FUNCTION_BLOCK ResetTrigger
  (* Standard: 61499-2 *)
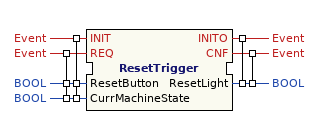
  EVENT_INPUT
    INIT WITH ResetButton, CurrMachineState;
    REQ WITH ResetButton, CurrMachineState;
  END_EVENT
  EVENT_OUTPUT
    INITO WITH ResetLight;
    CNF WITH ResetLight;
  END_EVENT
  VAR_INPUT
    ResetButton : BOOL;
    CurrMachineState : BOOL;
  END_VAR
  VAR_OUTPUT
    ResetLight : BOOL;
  END_VAR
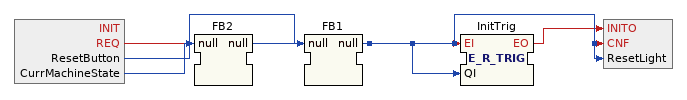
  FBS
    InitTrig : E_R_TRIG;
    FB1 : ;
    FB2 : ;
  END_FBS
  EVENT_CONNECTIONS
    FB1.null TO InitTrig.EI;
    FB2.null TO FB1.null;
    REQ TO FB2.null;
    InitTrig.EO TO INITO;
    FB1.null TO CNF;
  END_CONNECTIONS
  DATA_CONNECTIONS
    FB1.null TO InitTrig.QI;
    FB2.null TO FB1.null;
    FB1.null TO ResetLight;
    ResetButton TO FB1.null;
    CurrMachineState TO FB2.null;
  END_CONNECTIONS
END_FUNCTION_BLOCK
